RoboDK station: TRABAJO PRACTICO 5.rdk

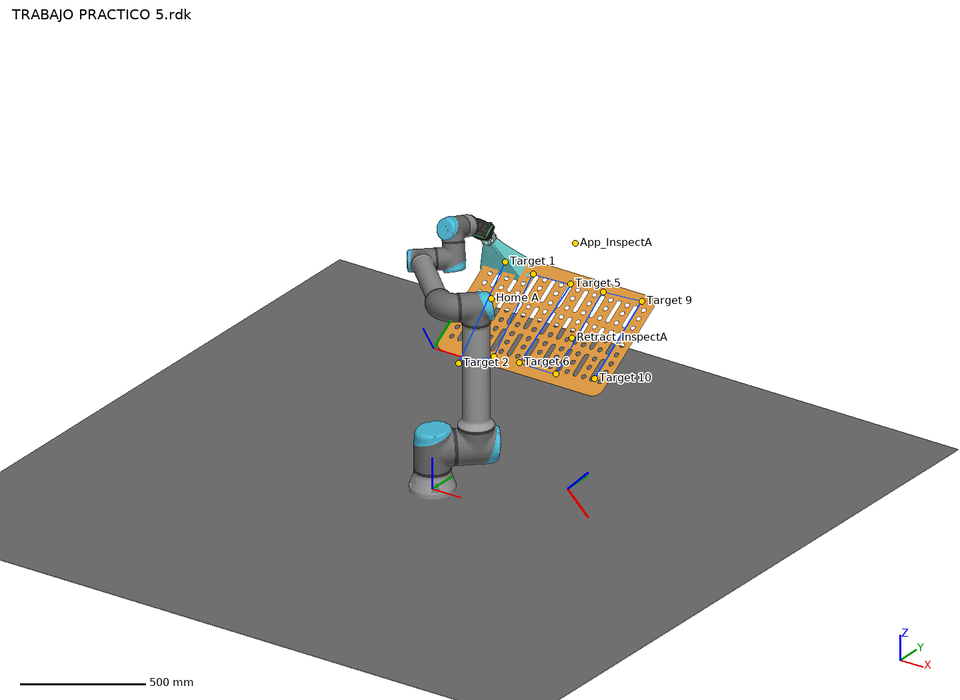
[picture v0: the station drawn from its stored meshes, robots at their saved joint values, targets as dots, program paths as lines]
Station TRABAJO PRACTICO 5 (saved by RoboDK 5.7.1). Poses are relative to the parent item; angles as X-Y-Z fixed-axis rotations.
Station parameters (name, value as stored): Palletizing Plugin
  - frame UR10e Base at (0, 0, 0) mm
    - robot UR10e: 6 axes, payload 10 kg, reach 1300 mm, repeatability 0.05 mm, weight 28.9 kg
        modified DH rows (alpha deg, a mm, theta deg, d mm): 0, 0, 0, 180.7; 90, 0, 180, 0; 0, 612.6, 0, 0; 0, 571.335, 0, 174.15; -90, 0, 0, 119.85; 90, 0, 180, 116.55
        joint limits [-360, -360, -360, -360, -360, -360] to [360, 360, 360, 360, 360, 360]; home [0, -90, -90, 0, 90, 0]; saved at [133.608, -90.438, -95.465, -17.191, 48.775, 195.696]
      - tool Camera 2, TCP at (0, -175.95, 321.06) mm, rotated rx 40 ry 0 rz 0 deg, size 215.7 x 276.1 x 372.4 mm
  - frame Frame Inspection A at (-380.72, 553.59, 295.24) mm, rotated rx 32.84 ry 0 rz 0 deg
    - object Inspection A at (0, 0, 0) mm, size 800 x 500 x 0 mm, geometry from Inspection A.step
    - folder Targets
    - target Target 1 (Cartesian target) at (79.2, 457.51, 5) mm, rotated rx -180 ry 0 rz 180 deg; joints [133.501, -90.589, -95.318, -17.151, 48.873, 195.641] of UR10e
    - target Target 2 (Cartesian target) at (141.75, -34.27, 5) mm, rotated rx 179.75 ry 0 rz 180 deg; joints [184.834, -41.161, -136.372, -107.963, 17.565, 286.215] of UR10e
    - target Target 3 (Cartesian target) at (270.26, 41.79, 5) mm, rotated rx 180 ry 0 rz 180 deg; joints [161.24, -38.764, -144.388, -40.681, 25.213, 220.978] of UR10e
    - target Target 4 (Cartesian target) at (224.75, 441.5, 5) mm, rotated rx -180 ry 0 rz 180 deg; joints [123.151, -84.661, -102.076, -13.507, 58.499, 190.907] of UR10e
    - target Target 5 (Cartesian target) at (403.61, 448.09, 5) mm, rotated rx -180 ry 0 rz 180 deg; joints [105.682, -83.563, -102.861, -11.357, 75.033, 184.735] of UR10e
    - target Target 6 (Cartesian target) at (390.7, 47.14, 5) mm, rotated rx 180 ry 0 rz 180 deg; joints [137.831, -39.235, -146.275, -19.19, 44.913, 198.041] of UR10e
    - target Target 7 (Cartesian target) at (568.48, 46.93, 5) mm, rotated rx -180 ry 0 rz 180 deg; joints [86.626, -56.24, -142.379, 1.432, 93.224, 179.004] of UR10e
    - target Target 8 (Cartesian target) at (554.74, 458.13, 5) mm, rotated rx -180 ry 0 rz 180 deg; joints [90.013, -86.994, -99.225, -10.94, 89.988, 180.004] of UR10e
    - target Target 9 (Cartesian target) at (750.45, 458.08, 25) mm, rotated rx 180 ry 0 rz 180 deg; joints [71.618, -93.897, -90.519, -13.607, 107.537, 174.401] of UR10e
    - target Target 10 (Cartesian target) at (750.21, 68.01, 25) mm, rotated rx 180 ry 0 rz 180 deg; joints [55.701, -74.55, -129.53, 3.586, 122.577, 168.622] of UR10e
    - target App_InspectA (Cartesian target) at (433.96, 543.11, 175.01) mm, rotated rx -172.24 ry 18.28 rz 174.82 deg; joints [115.29, -89.41, -72.94, -49.41, 49.41, 188.24] of UR10e
    - target Retract_InspectA (Cartesian target) at (750.21, 68.01, 315) mm, rotated rx 180 ry 0 rz -180 deg; joints [39.031, -62.165, -111.409, -32.544, 137.922, 160.003] of UR10e
    - target Home A (joint target) at (558.33, -45.25, 667.51) mm, rotated rx -180 ry 0 rz -180 deg; joints [90.932, -32.458, -85.483, -79.221, 89.109, 180.275] of UR10e
  - frame Frame Inspection B at (727.24, -100, 245.26) mm, rotated rx 0 ry 45.31 rz 0 deg
    - object Inspection B at (0, 0, 0) mm, size 202.5 x 1023.2 x 500 mm, geometry from Inspection B.step
  - frame World at (0, 0, 0) mm
    - object Floor at (0, 0, -7) mm, size 3000 x 3000 x 4.2 mm, geometry from Floor.step
  - folder InspectA
    - program InspectA (12 instructions, listed below)
    - program MainInspectA (5 instructions, listed below)
    - program App_InspectA (3 instructions, listed below)
    - program Retract_InspectA (3 instructions, listed below)
    - program GoHomeA (3 instructions, listed below)
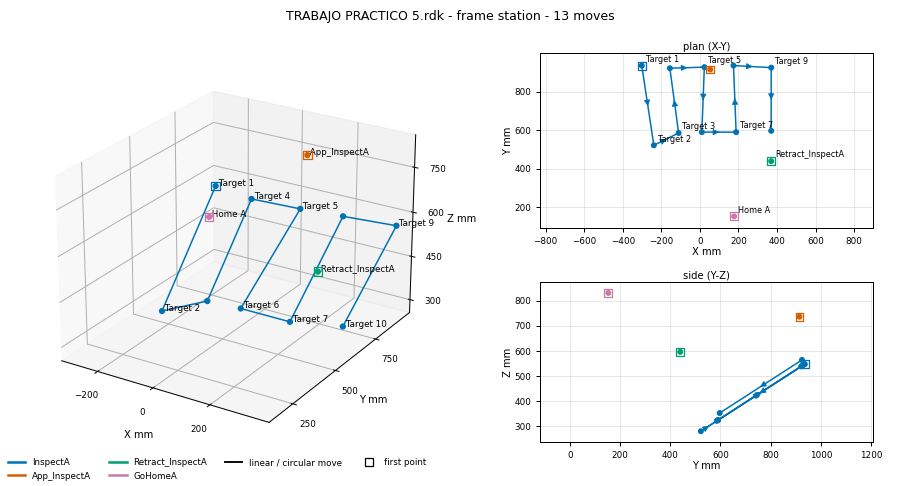
[picture p0: tool path of TRABAJO PRACTICO 5.rdk in frame station, 13 of 13 moves have a stored position in this frame; points joined in program order, loops and branches not executed]

--- program InspectA (robot UR10e) ---
  Est. Ref.: Frame Inspection A
  Est. herr: Camera 2
  MoveJ (Target 1)
  MoveL (Target 2)
  MoveL (Target 3)
  MoveL (Target 4)
  MoveL (Target 5)
  MoveL (Target 6)
  MoveL (Target 7)
  MoveL (Target 8)
  MoveL (Target 9)
  MoveL (Target 10)

--- program MainInspectA (robot UR10e) ---
  Llamar GoHomeA
  Llamar App_InspectA
  Llamar InspectA
  Llamar Retract_InspectA
  Llamar GoHomeA

--- program App_InspectA (robot UR10e) ---
  Est. Ref.: Frame Inspection A
  Est. herr: Camera 2
  MoveJ (App_InspectA)

--- program Retract_InspectA (robot UR10e) ---
  Est. Ref.: Frame Inspection A
  Est. herr: Camera 2
  MoveL (Retract_InspectA)

--- program GoHomeA (robot UR10e) ---
  Est. Ref.: Frame Inspection A
  Est. herr: Camera 2
  MoveJ (Home A)
